ABB RobotStudio station: VRM_project_Cervenka.rspag

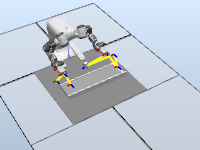
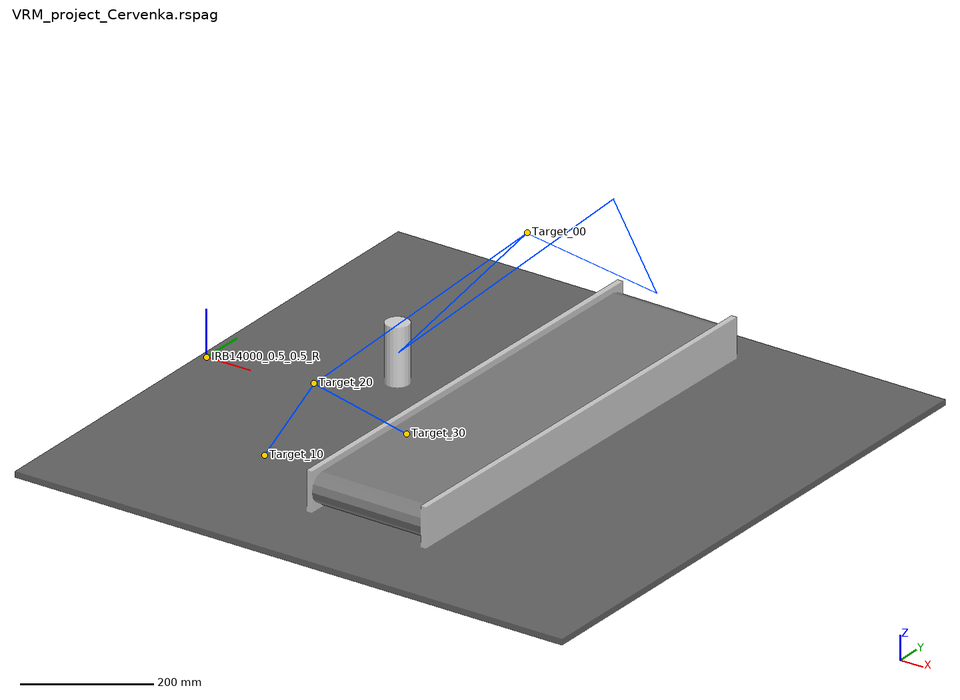
[picture v1: parts stored in the station drawn from their meshes, with robot base, taught points and paths (robot models come from the ABB library and are not in the file)]
--- station ---
Station Solution9 (saved by RobotStudio 21.4.9700.0)
Controller IRB14000
  mechanical unit ROB_R: IRB14000_0.5_0.5_R, 6 joints, base frame (0, 0, 0) mm
  mechanical unit ROB_R_7: IRB14000_0.5_0.5_R, 1 joints, base frame (0, 0, 0) mm
  mechanical unit ROB_L: IRB14000_0.5_0.5_L, 6 joints, base frame (0, 0, 0) mm
  mechanical unit ROB_L_7: IRB14000_0.5_0.5_L, 1 joints, base frame (0, 0, 0) mm
Layout (positions relative to the parent item):
  - IRB14000_0.5_0.5 [mechanism, from Robots\IRB14000_0.5_0.5__02.rslib] at (0, 0, 0) mm
  - IRB14000_0.5_0.5_R [mechanism, from Robots\IRB14000_0.5_0.5__02.rslib] at (0, 0, 0) mm; joint values [1.0732, -2.4606, -1.1122, 0.6063, 0.3644, 0.2549, 1.602] (rad or m)
  - IRB14000_0.5_0.5_L [mechanism, from Robots\IRB14000_0.5_0.5__02.rslib] at (0, 0, 0) mm; joint values [-0.8605, -2.3481, 1.1336, 0.3254, -0.2308, 0.5899, 1.1687] (rad or m)
  - Table [part], size 1000 x 1000 x 10 mm
  - Smart_Gripper_Servo_Fingers_2 [mechanism, from Tools\ABB_Smart_Gripper_Servo_Fingers.rslib] at (270.01, -267.25, 170.69) mm, rotated rx -90 ry 0 rz -90 deg; joint values [0.025] (rad or m)
  - Smart_Gripper_Servo_Fingers_3 [mechanism, from Tools\ABB_Smart_Gripper_Servo_Fingers.rslib] at (215.91, 366.18, 153.52) mm, rotated rx -90 ry 0 rz -90 deg; joint values [0.025] (rad or m)
  - Thing [part] at (632.38, 339.2, -0.2) mm, rotated rx 0 ry 0 rz -72.88 deg, size 40 x 39.9 x 100 mm
  - Attacher [smart component, from Components\Attacher.rslib]
      properties: Parent=Smart_Gripper_Servo_Fingers_2; Flange=0; Child=Thing; Mount=false; Offset=[0 0 0]; Orientation=[0 0 0]
  - Detacher [smart component, from Components\Detacher.rslib]
      properties: Child=Thing; KeepPosition=true
  - LinearMover [smart component, from Components\LinearMover.rslib]
      properties: Object=Thing; Direction=[0 0.001 0]; Speed=0.1; Reference=Global; ReferenceObject=(none)
  - LineSensor [smart component, from Components\LineSensor.rslib]
      properties: Start=[0.446335 0.372458 0.08392]; End=[0.659285 0.381354 0.083895]; Radius=0; SensedPart=(none); SensedPoint=[0 0 0]
    - _sensorPart_ [part], size 212.9 x 8.9 x 0 mm
  - Positioner [smart component, from Components\Positioner.rslib]
      properties: Object=Thing; Position=[0.215378 0.041769 0.001054]; Orientation=[0 0 0]; Reference=Global; ReferenceObject=(none)
  - Attacher_2 [smart component, from Components\Attacher.rslib] at (318.13, 59.56, 93.72) mm, rotated rx 0 ry 0 rz 72.88 deg
      properties: Parent=Smart_Gripper_Servo_Fingers_3; Flange=0; Child=Thing; Mount=false; Offset=[0 0 0]; Orientation=[0 0 0]
  - Detacher_2 [smart component, from Components\Detacher.rslib]
      properties: Child=Thing; KeepPosition=true
  - PoseMover_R [smart component, from Components\PoseMover.rslib] at (476.57, -525.07, 0) mm
      properties: Mechanism=Smart_Gripper_Servo_Fingers_2; Pose=1; Duration=1
  - PoseMover_R [smart component, from Components\PoseMover.rslib]
      properties: Mechanism=Smart_Gripper_Servo_Fingers_2; Pose=2; Duration=1
  - PoseMover_L [smart component, from Components\PoseMover.rslib] at (370.45, -539.65, 0) mm
      properties: Mechanism=Smart_Gripper_Servo_Fingers_3; Pose=2; Duration=1
  - PoseMover_L [smart component, from Components\PoseMover.rslib] at (476.57, -525.07, 0) mm
      properties: Mechanism=Smart_Gripper_Servo_Fingers_3; Pose=1; Duration=1
  - Conveyor [part] at (-329.87, -300.54, -144.17) mm, size 228.6 x 802.4 x 70.3 mm
Attachment: Smart_Gripper_Servo_Fingers_2 is attached to IRB14000_0.5_0.5_R / Link7
Attachment: Smart_Gripper_Servo_Fingers_3 is attached to IRB14000_0.5_0.5_L / Link7
Attachment: LinearMover is attached to Table
Attachment: Attacher_2 is attached to IRB14000_0.5_0.5_L / Link7
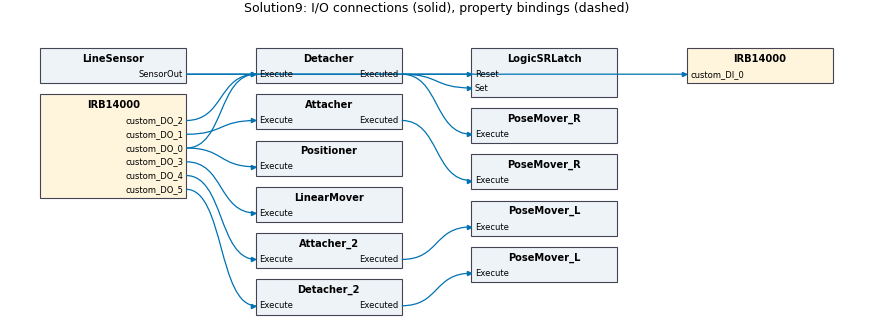
Station logic (signal -> signal, property => property):
  LineSensor.SensorOut -> LogicSRLatch.Reset
  IRB14000.custom_DO_2 -> Detacher.Execute
  IRB14000.custom_DO_1 -> Attacher.Execute
  Detacher.Executed -> LogicSRLatch.Set
  IRB14000.custom_DO_0 -> Positioner.Execute
  IRB14000.custom_DO_0 -> Detacher.Execute
  IRB14000.custom_DO_3 -> LinearMover.Execute
  LineSensor.SensorOut -> IRB14000.custom_DI_0
  IRB14000.custom_DO_4 -> Attacher_2.Execute
  IRB14000.custom_DO_5 -> Detacher_2.Execute
  Attacher.Executed -> PoseMover_R.Execute
  Detacher.Executed -> PoseMover_R.Execute
  Attacher_2.Executed -> PoseMover_L.Execute
  Detacher_2.Executed -> PoseMover_L.Execute

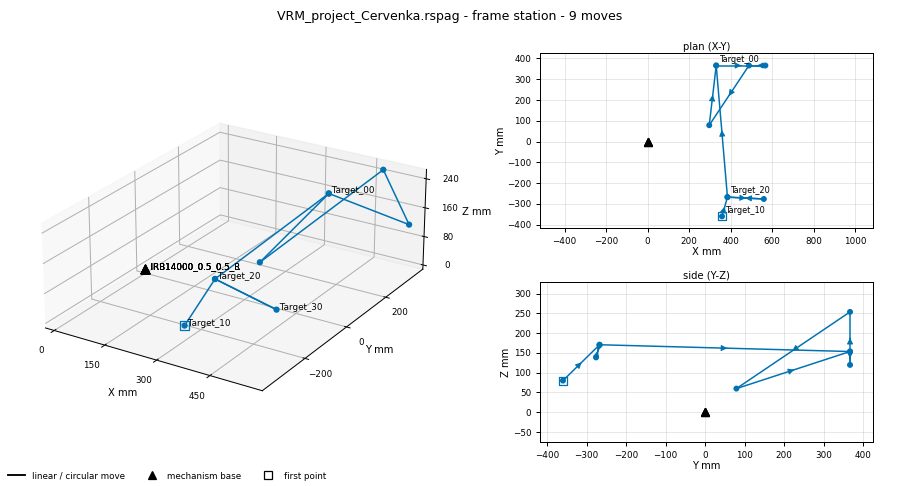
[picture p0: tool path of VRM_project_Cervenka.rspag in frame station, 9 of 9 moves have a stored position in this frame; points joined in program order, loops and branches not executed]
--- Backups/IRB14000/RAPID/TASK1/PROGMOD/CalibData.mod ---
MODULE CalibData
    PERS tooldata Servo:=[TRUE,[[0,0,114.2],[1,0,0,0]],[0.215,[8.7,12.3,49.2],[1,0,0,0],0.00021,0.00024,0.00009]];
    PERS tooldata Tooldata_1:=[TRUE,[[0,0,114.2],[1,0,0,0]],[0.215,[8.7,12.3,49.2],[1,0,0,0],0.00021,0.00024,0.00009]];
ENDMODULE

--- Backups/IRB14000/RAPID/TASK1/PROGMOD/Module1.mod ---
MODULE Module1
        CONST robtarget Target_10:=[[357.994922696,-359.830403815,79.958971591],[0.5,-0.5,0.5,-0.5],[1,0,1,4],[-101.964426493,9E+09,9E+09,9E+09,9E+09,9E+09]];
    CONST robtarget Target_20:=[[384.208016924,-267.247186969,170.693355338],[0.5,-0.5,0.5,-0.5],[1,0,1,4],[-101.964426493,9E+09,9E+09,9E+09,9E+09,9E+09]];
    CONST robtarget Target_30:=[[559.354511697,-276.222648897,138.649291138],[0.5,-0.5,0.5,-0.5],[1,0,1,4],[-101.964426493,9E+09,9E+09,9E+09,9E+09,9E+09]];
    CONST robtarget Target_40:=[[294.263,78.1,59.804],[0.704416026,-0.704416026,-0.061628417,0.061628417],[0,0,0,0],[-101.96443162,9E+09,9E+09,9E+09,9E+09,9E+09]];
!***********************************************************
    !
    ! Module:  Module1
    !
    ! Description:
    !   <Insert description here>
    !
    ! Author: suiti
    !
    ! Version: 1.0
    !
    !***********************************************************


    !***********************************************************
    !
    ! Procedure main
    !
    !   This is the entry point of your program
    !
    !***********************************************************
    PROC main()
        Path_10;
    ENDPROC
    PROC Path_10()
        PulseDO custom_DO_0; !reset
        MoveL Target_10,v1000,fine,Tooldata_1\WObj:=wobj0;
        PulseDO custom_DO_1; !attach
        WaitTime \InPos, 1;
        MoveL Target_20,v1000,fine,Tooldata_1\WObj:=wobj0;
        MoveL Target_30,v1000,fine,Tooldata_1\WObj:=wobj0;
        PulseDO custom_DO_2; !detach
        WaitTime 1;
        MoveL Target_20,v1000,fine,Tooldata_1\WObj:=wobj0;
        SetDO custom_DO_3, 1; ! run conveyor
        WaitUntil custom_DI_0 = 1; !sensor
        !off conveyor
        SetDO custom_DO_3,0;

    ENDPROC
ENDMODULE

--- Backups/IRB14000/RAPID/TASK2/PROGMOD/CalibData.mod ---
MODULE CalibData
    PERS tooldata Servo:=[TRUE,[[0,0,114.2],[1,0,0,0]],[0.215,[8.7,12.3,49.2],[1,0,0,0],0.00021,0.00024,0.00009]];
ENDMODULE

--- Backups/IRB14000/RAPID/TASK2/PROGMOD/Module1.mod ---
MODULE Module1
        CONST robtarget Target_00:=[[330.112611472,366.177,153.522304411],[0.5,-0.5,0.5,-0.5],[-1,0,1,4],[101.964427132,9E+09,9E+09,9E+09,9E+09,9E+09]];
    CONST robtarget Target_10:=[[566.737,366.177,119.744],[0.5,-0.5,0.5,-0.5],[-1,0,0,4],[101.964427132,9E+09,9E+09,9E+09,9E+09,9E+09]];
    CONST robtarget Target_20:=[[487.799658063,366.177,253.748829607],[0.5,-0.5,0.5,-0.5],[-1,1,0,4],[101.964427132,9E+09,9E+09,9E+09,9E+09,9E+09]];
    CONST robtarget Target_30:=[[296.557038398,78.806214933,59.803604774],[0.105248534,-0.105248534,0.69923011,-0.69923011],[-1,1,0,4],[101.964427132,9E+09,9E+09,9E+09,9E+09,9E+09]];
!***********************************************************
    !
    ! Module:  Module1
    !
    ! Description:
    !   <Insert description here>
    !
    ! Author: suiti
    !
    ! Version: 1.0
    !
    !***********************************************************


    !***********************************************************
    !
    ! Procedure main
    !
    !   This is the entry point of your program
    !
    !***********************************************************
    PROC main()
        Path_10;
    ENDPROC
    PROC Path_10()
        WaitUntil custom_DI_0 = 1 AND custom_DO_3 = 0;
        MoveL Target_00,v1000,z100,Servo\WObj:=wobj0;
        MoveL Target_10,v1000,fine,Servo\WObj:=wobj0;
        WaitTime \InPos, 1;
        PulseDO custom_DO_4;
        MoveL Target_20,v1000,fine,Servo\WObj:=wobj0;
        MoveL Target_30,v1000,fine,Servo\WObj:=wobj0;
        PulseDO custom_DO_5;
        MoveL Target_00, v1000, fine, Servo\WObj:=wobj0;
    ENDPROC
ENDMODULE

--- Backups/IRB14000/SYSPAR/EIO.cfg ---
EIO:CFG_1.0:6:1::
#
SYSSIG_IN:

      -Signal "Collision_Avoidance" -Action "CollAvoidance"
#
INDUSTRIAL_NETWORK:

      -Name "EtherNetIP" -Connection "Private Network"\
      -Label "EtherNet/IP Adapter Network"

      -Name "DeviceNet" -Label "DeviceNet Master/Slave Network" -Address "2"
#
EIO_CROSS:

      -Name "Cross_Signal_Lamp" -Res "Signal_Lamp" -Act1 "DRV1BRAKE"
#
EIO_SIGNAL_SAFELEVEL:

      -Name "FlangePowerSafeLevel" -ActionWhenStartup "Last"
#
DEVICENET_DEVICE:

      -Name "D652_10" -VendorName "ABB Robotics" -ProductName "24 VDC Unit"\
      -Address 10 -ProductCode 26 -DeviceType 7 -ConnectionType "COS"\
      -OutputSize 2 -InputSize 2
#
DEVICENET_INTERNAL_DEVICE:

      -Name "DN_Internal_Device" -VendorName "ABB Robotics"\
      -ProductName "DeviceNet Internal Slave Device"
#
ETHERNETIP_INTERNAL_DEVICE:

      -Name "EN_Internal_Device" -VendorName "ABB Robotics"\
      -ProductName "EtherNet/IP Internal Adapter Device"
#
EIO_SIGNAL:

      -Name "custom_DI_0" -SignalType "DI" -Device "D652_10" -DeviceMap "0"

      -Name "custom_DI_1" -SignalType "DI" -Device "D652_10" -DeviceMap "1"

      -Name "custom_DI_2" -SignalType "DI" -Device "D652_10" -DeviceMap "2"

      -Name "custom_DI_3" -SignalType "DI" -Device "D652_10" -DeviceMap "3"

      -Name "custom_DI_4" -SignalType "DI" -Device "D652_10" -DeviceMap "4"

      -Name "custom_DI_5" -SignalType "DI" -Device "D652_10" -DeviceMap "5"

      -Name "custom_DI_6" -SignalType "DI" -Device "D652_10" -DeviceMap "6"

      -Name "custom_DI_7" -SignalType "DI" -Device "D652_10" -DeviceMap "7"

      -Name "custom_DO_0" -SignalType "DO" -Device "D652_10" -DeviceMap "0"

      -Name "custom_DO_1" -SignalType "DO" -Device "D652_10" -DeviceMap "1"

      -Name "custom_DO_2" -SignalType "DO" -Device "D652_10" -DeviceMap "2"

      -Name "custom_DO_3" -SignalType "DO" -Device "D652_10" -DeviceMap "3"

      -Name "custom_DO_4" -SignalType "DO" -Device "D652_10" -DeviceMap "4"

      -Name "custom_DO_5" -SignalType "DO" -Device "D652_10" -DeviceMap "5"

      -Name "custom_DO_6" -SignalType "DO" -Device "D652_10" -DeviceMap "6"

      -Name "custom_DO_7" -SignalType "DO" -Device "D652_10" -DeviceMap "7"

      -Name "hall_sensor_joint_1" -SignalType "DI" -Device "D652_10"\
      -DeviceMap "8"

      -Name "hall_sensor_joint_2" -SignalType "DI" -Device "D652_10"\
      -DeviceMap "9"

      -Name "hall_sensor_joint_3" -SignalType "DI" -Device "D652_10"\
      -DeviceMap "11"

      -Name "hall_sensor_joint_4" -SignalType "DI" -Device "D652_10"\
      -DeviceMap "12"

      -Name "hall_sensor_joint_5" -SignalType "DI" -Device "D652_10"\
      -DeviceMap "13"

      -Name "hall_sensor_joint_6" -SignalType "DI" -Device "D652_10"\
      -DeviceMap "14"

      -Name "hall_sensor_joint_7" -SignalType "DI" -Device "D652_10"\
      -DeviceMap "10"

      -Name "hall_sensor_24V_ROB_R" -SignalType "DO" -Device "D652_10"\
      -DeviceMap "8"

      -Name "hall_sensor_24V_ROB_L" -SignalType "DO" -Device "D652_10"\
      -DeviceMap "9"

      -Name "flange_24V_ROB_R" -SignalType "DO" -Device "D652_10"\
      -DeviceMap "10" -SafeLevel "FlangePowerSafeLevel"

      -Name "flange_24V_ROB_L" -SignalType "DO" -Device "D652_10"\
      -DeviceMap "11" -SafeLevel "FlangePowerSafeLevel"

      -Name "Signal_Lamp" -SignalType "DO" -Device "D652_10" -DeviceMap "12"

      -Name "Collision_Avoidance" -SignalType "DO" -Access "All" -Default 1
